FUNCTION_BLOCK ControlFBD_Sequence
VAR_INPUT
	 mxAutoRunOk     : BOOL;
    mxAutoModeReady : BOOL;
    ixSliderAout    : BOOL;
	ixSliderAin    : BOOL;
    ixDrillDown     : BOOL;
    ixDrillUp       : BOOL;
    ixSliderBout    : BOOL;
    ixSliderBin     : BOOL;
END_VAR
VAR_OUTPUT
	mxAutoAout      : BOOL;
    mxAutoDrillDown : BOOL;
    mxAutoDrillUp   : BOOL;
    mxAutoBout      : BOOL;
    mxAutoBin       : BOOL;
    mxAutoAin       : BOOL;
END_VAR
VAR
	miSeq : STATES := STATES.init;
END_VAR

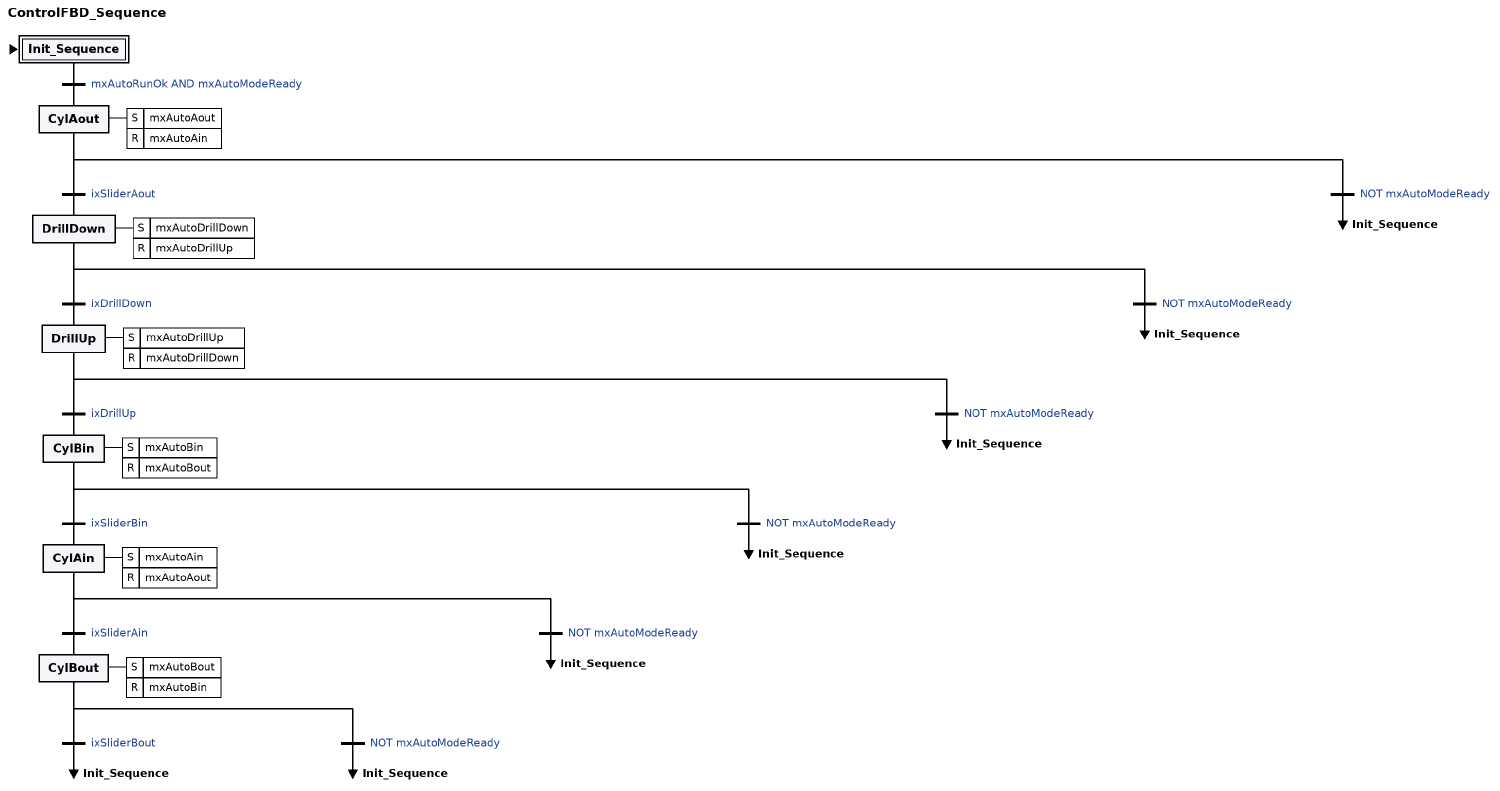
INITIAL_STEP Init_Sequence:
END_STEP
TRANSITION FROM Init_Sequence TO CylAout
    := mxAutoRunOk AND mxAutoModeReady;
END_TRANSITION
STEP CylAout:
    mxAutoAout(S);
    mxAutoAin(R);
END_STEP
TRANSITION FROM CylAout TO DrillDown
    := ixSliderAout;
END_TRANSITION
STEP DrillDown:
    mxAutoDrillDown(S);
    mxAutoDrillUp(R);
END_STEP
TRANSITION FROM DrillDown TO DrillUp
    := ixDrillDown;
END_TRANSITION
STEP DrillUp:
    mxAutoDrillUp(S);
    mxAutoDrillDown(R);
END_STEP
TRANSITION FROM DrillUp TO CylBin
    := ixDrillUp;
END_TRANSITION
STEP CylBin:
    mxAutoBin(S);
    mxAutoBout(R);
END_STEP
TRANSITION FROM CylBin TO CylAin
    := ixSliderBin;
END_TRANSITION
STEP CylAin:
    mxAutoAin(S);
    mxAutoAout(R);
END_STEP
TRANSITION FROM CylAin TO CylBout
    := ixSliderAin;
END_TRANSITION
STEP CylBout:
    mxAutoBout(S);
    mxAutoBin(R);
END_STEP
TRANSITION FROM CylBout TO Init_Sequence
    := ixSliderBout;
END_TRANSITION
TRANSITION FROM CylBout TO Init_Sequence
    := NOT mxAutoModeReady;
END_TRANSITION
TRANSITION FROM CylAin TO Init_Sequence
    := NOT mxAutoModeReady;
END_TRANSITION
TRANSITION FROM CylBin TO Init_Sequence
    := NOT mxAutoModeReady;
END_TRANSITION
TRANSITION FROM DrillUp TO Init_Sequence
    := NOT mxAutoModeReady;
END_TRANSITION
TRANSITION FROM DrillDown TO Init_Sequence
    := NOT mxAutoModeReady;
END_TRANSITION
TRANSITION FROM CylAout TO Init_Sequence
    := NOT mxAutoModeReady;
END_TRANSITION

END_FUNCTION_BLOCK

(* stored: Version 1.1.0.1
   POU ControlFBD_Sequence: Id {907a818c-f43f-43a4-8f4e-946302b3e32d}, SpecialFunc None *)
